// TwinCAT 3 PLC project ph_lv1_Motion
// Title: tclib_ph_lv1_motion
// Company: Poh
// Author: Poh
// ProjectVersion: 0.1.3.0
// ProgramVersion: 3.1.4020.1
// libraries:
//   Tc2_MC2, * (Beckhoff Automation GmbH)
//   tclib_ph_lv0, * (Poh)
// project tree:
//   Lv1_Motion/Class/ C_ACTUATION.TcPOU, C_ACTUATION_EXT_HOMING.TcPOU
//   Lv1_Motion/Data/ S_ACTUATION_LINK.TcDUT
//   Lv1_Motion/Interface/ IFC_ACTUATION.TcIO
// (motion and I/O tree: see PLC project ph_lv0)
// real-time tasks:
//   TASK PlcTask: cycle T#10ms, priority 20, ADS port 350
//   TASK Fast: cycle T#3ms, priority 1, ADS port 351

// ---- Lv1_Motion/Data/S_ACTUATION_LINK.TcDUT
TYPE S_ACTUATION_LINK :
STRUCT
	HARDWARE_ERROR_ID 	: UDINT;
	CALIBRATION_SENSOR	: BOOL;
	LIMIT_MINUS 		: BOOL;
	LIMIT_PLUS			: BOOL;
END_STRUCT
END_TYPE

// ---- Lv1_Motion/Interface/IFC_ACTUATION.TcIO
INTERFACE IFC_ACTUATION

PROPERTY Acceleration : LREAL
GET
END_GET
SET
END_SET
END_PROPERTY

PROPERTY Axis_Id : UDINT
GET
END_GET
END_PROPERTY

(*
	Y:2016		M:05	D:20
	D: Initiates the manual motion of the actuation device. Keep the method running for as long as manual motion is required. Terminate manual motion by calling the opposite method.
*)
METHOD Begin_Jog : RETURN_CODE
VAR_INPUT
	Towards_Positive : BOOL;
END_VAR
END_METHOD

PROPERTY Calibrate_At_Minus : BOOL
GET
END_GET
SET
END_SET
END_PROPERTY

PROPERTY Controller_Override : LREAL
GET
END_GET
SET
END_SET
END_PROPERTY

PROPERTY Current_Position : LREAL
GET
END_GET
END_PROPERTY

PROPERTY Current_Velocity : LREAL
GET
END_GET
END_PROPERTY

PROPERTY Deceleration : LREAL
GET
END_GET
SET
END_SET
END_PROPERTY

(*
	Y:2016		M:05	D:20
	D: Sets the actuation device in a de-energised state, and disable travel on both directions.
*)
METHOD Disable : RETURN_CODE
VAR_INPUT
END_VAR
END_METHOD

PROPERTY Enable : BOOL
GET
END_GET
SET
END_SET
END_PROPERTY

(*
	Y:2016		M:05	D:20
	D: Sets the actuation device in a energised state, and enable travel on both directions.
*)
METHOD Enable_All : RETURN_CODE
VAR_INPUT
END_VAR
END_METHOD

PROPERTY Enable_Bw : BOOL
GET
END_GET
SET
END_SET
END_PROPERTY

PROPERTY Enable_Fw : BOOL
GET
END_GET
SET
END_SET
END_PROPERTY

(*
	Y:2016		M:05	D:20
	D: Terminates the manual motion of the actuation device.
*)
METHOD End_Jog : RETURN_CODE
VAR_INPUT
END_VAR
END_METHOD

(*
	Y:2016		M:05	D:20
	D: Halts the actuation device.
*)
METHOD Halt : RETURN_CODE
VAR_INPUT
END_VAR
END_METHOD

(*
	Y:2016		M:05	D:20
	D: Initiates the homing sequence for the actuation device. Configure the homing behavior via the class's properties.
*)
METHOD Home : RETURN_CODE
VAR_INPUT
END_VAR
END_METHOD

PROPERTY Home_To_Limit : BOOL
GET
END_GET
SET
END_SET
END_PROPERTY

PROPERTY Is_Disabled : BOOL
GET
END_GET
END_PROPERTY

PROPERTY Is_Error : BOOL
GET
END_GET
END_PROPERTY

PROPERTY Is_Moving : BOOL
GET
END_GET
END_PROPERTY

PROPERTY Jerk : LREAL
GET
END_GET
SET
END_SET
END_PROPERTY

(*
	Y:2016		M:05	D:20
	D: Sets the actuation in motion along a direction.
*)
METHOD Move_Along : RETURN_CODE
VAR_INPUT
	Positive_Direction : BOOL;
END_VAR
END_METHOD

(*
	Y:2016		M:05	D:20
	D: Sets the actuation device in motion for a specified distance.
*)
METHOD Move_By : RETURN_CODE
VAR_INPUT
	//User defined distance to travel. Can be + or -
		Distance : LREAL;
END_VAR
END_METHOD

(*
	Y:2016		M:05	D:20
	D: Sets the actuation in motion to the target position.
*)
METHOD Move_To : RETURN_CODE
VAR_INPUT
	//User defined position to travel. Can be + or -
		POSITION : LREAL;
END_VAR
END_METHOD

(*
	Y:2016		M:05	D:20
	D: Resets the actuation device of any errors. Actuation device currently in motion will be halted.
*)
METHOD Reset : RETURN_CODE
VAR_INPUT
END_VAR
END_METHOD

PROPERTY Velocity : LREAL
GET
END_GET
SET
END_SET
END_PROPERTY

END_INTERFACE

// ---- Lv1_Motion/Class/C_ACTUATION.TcPOU
(*
	Y:2016		M:05		D:20
	T:CLASS		N:ACTUATION
	D:Class object for plc motion projects. Contains all basic necessary methods for movement. The default behavior is to home to negative limit.
*)
FUNCTION_BLOCK C_ACTUATION IMPLEMENTS IFC_ACTUATION
VAR_INPUT
END_VAR
VAR_OUTPUT
END_VAR
VAR
	//SOFTWARAE PDO LINK
		_AXIS : AXIS_REF;	
	//HARDWARE PDO LINK
		_HARDWARE_LINK	AT %I*	: S_ACTUATION_LINK;
	//MOTION MODULES
		_M_POWER 	: MC_POWER;
		_M_RESET 	: MC_RESET;
		_M_MOVEA 	: MC_MOVEABSOLUTE;
		_M_MOVER 	: MC_MOVERELATIVE;
		_M_HOME		: MC_HOME;
		_M_HALT		: MC_HALT;
		_M_MOVEEL	: MC_MoveVelocity;
		_M_JOG		: MC_JOG;
	//DYNAMICS
		_VELOCITY 		: LREAL := 10;
		_ACCELERATION 	: LREAL := 0;
		_DECELERATION 	: LREAL := 0;
		_JERK 			: LREAL := 0;
	//
		_HOME_TO_LIMIT	: BOOL := TRUE;
		_HOME_TO_MINUS	: BOOL := TRUE;
END_VAR

PROPERTY Acceleration : LREAL
GET
Acceleration := _ACCELERATION;
END_GET
SET
_ACCELERATION := ABS(Acceleration);
END_SET
END_PROPERTY

PROPERTY Axis_Id : UDINT
GET
Axis_Id := _AXIS.NcToPlc.AxisId;
END_GET
END_PROPERTY

(*
	Y:2016		M:05	D:20
	D: Initiates the manual motion of the actuation device. Keep the method running for as long as manual motion is required. Terminate manual motion by calling the opposite method.
*)
METHOD Begin_Jog : RETURN_CODE
VAR_INPUT
	Towards_Positive : BOOL;
END_VAR
_M_JOG(
	Axis:= _AXIS, 
	JogForward:= Towards_Positive, 
	JogBackwards:= NOT Towards_Positive, 
	Mode:= MC_JOGMODE_CONTINOUS, 
	Velocity:= _VELOCITY, 
	Acceleration:= _ACCELERATION, 
	Deceleration:= _DECELERATION, 
	Jerk:= _JERK);
IF _M_JOG.Error THEN
	Begin_Jog := ph_lv0.LV0_RETURNCODE.RETURN_ERROR;
ELSIF _M_JOG.CommandAborted THEN
	Begin_Jog := ph_lv0.LV0_RETURNCODE.RETURN_ERROR + 1;
ELSIF _M_JOG.Active THEN
	Begin_Jog := ph_lv0.LV0_RETURNCODE.RETURN_SUCCESS;
ELSE
	Begin_Jog := ph_lv0.LV0_RETURNCODE.RETURN_BUSY;
END_IF
END_METHOD

PROPERTY Calibrate_At_Minus : BOOL
GET
Calibrate_At_Minus := _HOME_TO_MINUS;
END_GET
SET
_HOME_TO_MINUS := Calibrate_At_Minus;
END_SET
END_PROPERTY

PROPERTY Controller_Override : LREAL
GET
VAR
	_FACTOR : LREAL := 1000000;
END_VAR
Controller_Override := (_AXIS.PlcToNc.Override / _FACTOR) * 100.0;
END_GET
SET
VAR
	_BUFFER : LREAL;
	_FACTOR : LREAL := 1000000;
END_VAR
IF Controller_Override > 100.0 THEN
	_BUFFER := 100.0;
ELSIF Controller_Override < 0.0 THEN 
	_BUFFER := 0.0;
ELSE 
	_BUFFER := Controller_Override;
END_IF
_AXIS.PlcToNc.Override := LREAL_TO_UDINT((_BUFFER/100.0) * _FACTOR);
END_SET
END_PROPERTY

PROPERTY Current_Position : LREAL
GET
Current_Position := _AXIS.NcToPlc.ActPos;
END_GET
END_PROPERTY

PROPERTY Current_Velocity : LREAL
GET
Current_Velocity := _AXIS.NcToPlc.ActVelo;
END_GET
END_PROPERTY

PROPERTY Deceleration : LREAL
GET
Deceleration := _DECELERATION;
END_GET
SET
_DECELERATION := ABS(Deceleration);
END_SET
END_PROPERTY

(*
	Y:2016		M:05	D:20
	D: Sets the actuation device in a de-energised state, and disable travel on both directions.
*)
METHOD Disable : RETURN_CODE
VAR_INPUT
END_VAR
_M_POWER(
	Axis:= _AXIS, 
	Enable:= FALSE, 
	Enable_Positive:= FALSE, 
	Enable_Negative:= FALSE, 
	Override:= 0 );

IF _M_POWER.Error THEN
	Disable := ph_lv0.LV0_RETURNCODE.RETURN_ERROR;
ELSIF NOT _M_POWER.Status THEN
	Disable := ph_lv0.LV0_RETURNCODE.RETURN_SUCCESS;
ELSE
	Disable := ph_lv0.LV0_RETURNCODE.RETURN_BUSY;
END_IF
END_METHOD

PROPERTY Enable : BOOL
GET
Enable := _AXIS.PlcToNc.ControlDWord.0;
END_GET
SET
_AXIS.PlcToNc.ControlDWord.0 := Enable;
END_SET
END_PROPERTY

(*
	Y:2016		M:05	D:20
	D: Sets the actuation device in a energised state, and enable travel on both directions.
*)
METHOD Enable_All : RETURN_CODE
VAR_INPUT
END_VAR
_M_POWER(
	Axis:= _AXIS, 
	Enable:= TRUE, 
	Enable_Positive:= TRUE, 
	Enable_Negative:= TRUE, 
	Override:= 100 );

IF _M_POWER.Error THEN
	Enable_All := ph_lv0.LV0_RETURNCODE.RETURN_ERROR;
ELSIF _M_POWER.Status THEN
	Enable_All := ph_lv0.LV0_RETURNCODE.RETURN_SUCCESS;
ELSE
	Enable_All := ph_lv0.LV0_RETURNCODE.RETURN_BUSY;
END_IF
END_METHOD

PROPERTY Enable_Bw : BOOL
GET
Enable_Bw := _AXIS.PlcToNc.ControlDWord.2;
END_GET
SET
_AXIS.PlcToNc.ControlDWord.2 := Enable_Bw;
END_SET
END_PROPERTY

PROPERTY Enable_Fw : BOOL
GET
Enable_Fw := _AXIS.PlcToNc.ControlDWord.1;
END_GET
SET
_AXIS.PlcToNc.ControlDWord.1 := Enable_Fw;
END_SET
END_PROPERTY

(*
	Y:2016		M:05	D:20
	D: Terminates the manual motion of the actuation device.
*)
METHOD End_Jog : RETURN_CODE
VAR_INPUT
END_VAR
_M_JOG(
	Axis:= _AXIS, 
	JogForward:= FALSE, 
	JogBackwards:= FALSE);
IF _M_JOG.Error THEN
	End_Jog := ph_lv0.LV0_RETURNCODE.RETURN_ERROR;
ELSIF _M_JOG.CommandAborted THEN
	End_Jog := ph_lv0.LV0_RETURNCODE.RETURN_ERROR + 1;
ELSIF _M_JOG.Done THEN
	End_Jog := ph_lv0.LV0_RETURNCODE.RETURN_SUCCESS;
ELSE
	End_Jog := ph_lv0.LV0_RETURNCODE.RETURN_BUSY;
END_IF
END_METHOD

(*
	Y:2016		M:05	D:20
	D: Halts the actuation device.
*)
METHOD Halt : RETURN_CODE
VAR_INPUT
END_VAR
_M_HALT(
	Axis:= _AXIS, 
	Execute:= TRUE, 
	Deceleration:= _DECELERATION, 
	Jerk:= _JERK);
IF _M_HALT.Error THEN
	_M_HALT(
		Axis:=_AXIS,
		Execute:=FALSE);
	Halt:=ph_lv0.LV0_RETURNCODE.RETURN_ERROR;
ELSIF _M_HALT.CommandAborted THEN
	_M_HALT(
		Axis:=_AXIS,
		Execute:=FALSE);
	Halt:=ph_lv0.LV0_RETURNCODE.RETURN_ERROR + 1;
ELSIF _M_HALT.Done THEN
	_M_HALT(
		Axis:=_AXIS,
		Execute:=FALSE);
	Halt:=ph_lv0.LV0_RETURNCODE.RETURN_SUCCESS;
ELSE
	Halt:=ph_lv0.LV0_RETURNCODE.RETURN_BUSY;
END_IF
END_METHOD

(*
	Y:2016		M:05	D:20
	D: Initiates the homing sequence for the actuation device. Configure the homing behavior via the class's properties.
*)
METHOD Home : RETURN_CODE
VAR_INPUT
END_VAR
VAR
	_CALIBRATION_FLAG : BOOL;
END_VAR
IF _HOME_TO_LIMIT THEN
	IF _HOME_TO_MINUS THEN
		_CALIBRATION_FLAG := THIS^._HARDWARE_LINK.LIMIT_MINUS;
	ELSE
		_CALIBRATION_FLAG := THIS^._HARDWARE_LINK.LIMIT_PLUS;
	END_IF
ELSE
	_CALIBRATION_FLAG := THIS^._HARDWARE_LINK.CALIBRATION_SENSOR;
END_IF
_M_HOME(
	Axis:= _AXIS, 
	Execute:= TRUE, 
	bCalibrationCam:= _CALIBRATION_FLAG);
IF _M_HOME.Error THEN
	_M_HOME(
		Axis:= _AXIS, 
		Execute:= FALSE);
	Home := ph_lv0.LV0_RETURNCODE.RETURN_ERROR;
ELSIF _M_HOME.CommandAborted THEN
	_M_HOME(
		Axis:= _AXIS, 
		Execute:= FALSE);
	Home := ph_lv0.LV0_RETURNCODE.RETURN_ERROR + 1;
ELSIF _M_HOME.Done THEN
	_M_HOME(
		Axis:= _AXIS, 
		Execute:= FALSE);
	Home := ph_lv0.LV0_RETURNCODE.RETURN_SUCCESS;
ELSE
	Home := ph_lv0.LV0_RETURNCODE.RETURN_BUSY;
END_IF
END_METHOD

PROPERTY Home_To_Limit : BOOL
GET
Home_To_Limit := _HOME_TO_LIMIT;
END_GET
SET
_HOME_TO_LIMIT := Home_To_Limit;
END_SET
END_PROPERTY

PROPERTY Is_Disabled : BOOL
GET
_AXIS.ReadStatus();
Is_Disabled := _AXIS.Status.Disabled;
END_GET
END_PROPERTY

PROPERTY Is_Error : BOOL
GET
_AXIS.ReadStatus();
Is_Error := _AXIS.Status.Error;
END_GET
END_PROPERTY

PROPERTY Is_Moving : BOOL
GET
_AXIS.ReadStatus();
Is_Moving := _AXIS.Status.Moving;
END_GET
END_PROPERTY

PROPERTY Jerk : LREAL
GET
Jerk := _JERK;
END_GET
SET
_JERK := ABS(Jerk);
END_SET
END_PROPERTY

(*
	Y:2016		M:05	D:20
	D: Sets the actuation in motion along a direction.
*)
METHOD Move_Along : RETURN_CODE
VAR_INPUT
	Positive_Direction : BOOL;
END_VAR
VAR
	_DIRECTION : MC_Direction;
END_VAR
IF Positive_Direction THEN
	_DIRECTION := MC_Direction.MC_Positive_Direction;
ELSE
	_DIRECTION := MC_Direction.MC_Negative_Direction;
END_IF
_M_MOVEEL(
	Axis:= _AXIS, 
	Execute:= TRUE, 
	Velocity:= _VELOCITY, 
	Acceleration:= _ACCELERATION, 
	Deceleration:= _DECELERATION, 
	Jerk:= _JERK, 
	Direction:= _DIRECTION);
IF _M_MOVEEL.Error THEN
	_M_MOVEEL(
		Axis:= _AXIS, 
		Execute:= FALSE); 
	Move_Along := ph_lv0.LV0_RETURNCODE.RETURN_ERROR;
ELSIF _M_MOVEEL.CommandAborted THEN
	_M_MOVEEL(
		Axis:= _AXIS, 
		Execute:= FALSE);
	Move_Along := ph_lv0.LV0_RETURNCODE.RETURN_ERROR + 1;
ELSIF _M_MOVEEL.InVelocity THEN
	_M_MOVEEL(
		Axis:= _AXIS, 
		Execute:= FALSE);
	Move_Along := ph_lv0.LV0_RETURNCODE.RETURN_SUCCESS;
ELSE
	Move_Along := ph_lv0.LV0_RETURNCODE.RETURN_BUSY;
END_IF
END_METHOD

(*
	Y:2016		M:05	D:20
	D: Sets the actuation device in motion for a specified distance.
*)
METHOD Move_By : RETURN_CODE
VAR_INPUT
	//User defined distance to travel. Can be + or -
		Distance : LREAL;
END_VAR
_M_MOVER(
	Axis:= _AXIS, 
	Execute:= TRUE, 
	Distance:= Distance, 
	Velocity:= _VELOCITY, 
	Acceleration:= _ACCELERATION, 
	Deceleration:= _DECELERATION, 
	Jerk:= _JERK);
	
IF _M_MOVER.Error THEN
	_M_MOVER(
		Axis:= _AXIS, 
		Execute:= FALSE);
	Move_By := ph_lv0.LV0_RETURNCODE.RETURN_ERROR;
ELSIF _M_MOVER.CommandAborted THEN
	_M_MOVER(
		Axis:= _AXIS, 
		Execute:= FALSE);
	Move_By := ph_lv0.LV0_RETURNCODE.RETURN_ERROR + 1;
ELSIF _M_MOVER.Done THEN
	_M_MOVER(
		Axis:= _AXIS, 
		Execute:= FALSE);
	Move_By := ph_lv0.LV0_RETURNCODE.RETURN_SUCCESS;
ELSE
	Move_By := ph_lv0.LV0_RETURNCODE.RETURN_BUSY;	
END_IF
END_METHOD

(*
	Y:2016		M:05	D:20
	D: Sets the actuation in motion to the target position.
*)
METHOD Move_To : RETURN_CODE
VAR_INPUT
	//User defined position to travel. Can be + or -
		POSITION : LREAL;
END_VAR
_M_MOVEA(
	Axis:= _AXIS, 
	Execute:= TRUE, 
	Position:= POSITION, 
	Velocity:= _VELOCITY, 
	Acceleration:= _ACCELERATION, 
	Deceleration:= _DECELERATION, 
	Jerk:= _JERK);
IF _M_MOVEA.Error THEN
	_M_MOVEA(
		Axis:= _AXIS, 
		Execute:= FALSE);
	Move_To := ph_lv0.LV0_RETURNCODE.RETURN_ERROR;
ELSIF _M_MOVEA.CommandAborted THEN
	_M_MOVEA(
		Axis:= _AXIS, 
		Execute:= FALSE);
	Move_To := ph_lv0.LV0_RETURNCODE.RETURN_ERROR + 1;
ELSIF _M_MOVEA.Done THEN
	_M_MOVEA(
		Axis:= _AXIS, 
		Execute:= FALSE);
	Move_To := ph_lv0.LV0_RETURNCODE.RETURN_SUCCESS;
ELSE
	Move_To := ph_lv0.LV0_RETURNCODE.RETURN_BUSY;	
END_IF
END_METHOD

(*
	Y:2016		M:05	D:20
	D: Resets the actuation device of any errors. Actuation device currently in motion will be halted.
*)
METHOD Reset : RETURN_CODE
VAR_INPUT
END_VAR
//RESET OTHER FUNCTION BLOCKS
	_M_MOVEA(
		Axis:= _AXIS,
		Execute:= FALSE);
	_M_MOVER(
		Axis:= _AXIS, 
		Execute:= FALSE);
	_M_MOVEEL(
		Axis:= _AXIS, 
		Execute:= FALSE);
	_M_HALT(
		Axis:= _AXIS, 
		Execute:= FALSE);
	_M_HOME(
		Axis:= _AXIS, 
		Execute:= FALSE);
//EXECUTE RESET
	_M_RESET(
		Axis:= _AXIS, 
		Execute:= TRUE);
	IF _M_RESET.Error THEN
		_M_RESET(
			Axis:= _AXIS, 
			Execute:= FALSE);
		Reset := ph_lv0.LV0_RETURNCODE.RETURN_ERROR;
	ELSIF _M_RESET.Done AND NOT _M_RESET.Busy THEN
		_M_RESET(
			Axis:= _AXIS, 
			Execute:= FALSE);
		Reset := ph_lv0.LV0_RETURNCODE.RETURN_SUCCESS;
	ELSE
		Reset := ph_lv0.LV0_RETURNCODE.RETURN_BUSY;	
	END_IF
END_METHOD

PROPERTY Velocity : LREAL
GET
Velocity := _VELOCITY;
END_GET
SET
_VELOCITY := ABS(Velocity);
END_SET
END_PROPERTY

END_FUNCTION_BLOCK

// ---- Lv1_Motion/Class/C_ACTUATION_EXT_HOMING.TcPOU
FUNCTION_BLOCK C_ACTUATION_EXT_HOMING EXTENDS C_ACTUATION
VAR_INPUT
END_VAR
VAR_OUTPUT
END_VAR
VAR
	_HardStopCalibration	: BOOL := FALSE;
	_HardStopTol			: LREAL := 5.0;
END_VAR

PROPERTY Calibrate_At_Hardstop : BOOL
GET
Calibrate_At_Hardstop := _HardStopCalibration;
END_GET
SET
_HardStopCalibration := Calibrate_At_Hardstop;
END_SET
END_PROPERTY

PROPERTY Hardstop_Tolerance : LREAL
GET
Hardstop_Tolerance := _HardStopTol;
END_GET
SET
 _HardStopTol := Hardstop_Tolerance;
END_SET
END_PROPERTY

{attribute '''NORMAL__COMMENT' := '
	Y:2016		M:05	D:20
	D: Initiates the homing sequence for the actuation device. Configure the homing behavior via the class's properties.
'}
(*
	Y:2016		M:05	D:20
	D: Initiates the homing sequence for the actuation device. Configure the homing behavior via the class's properties.
*)
(*
	Y:2016		M:06	D:03
	D: Initiates the homing sequence for the actuation device. Configure the homing behavior via the class's properties.
	EXT: Uses the Use_Hard_Stop option to calibrate the homing sequence
*)
METHOD Home : ph_lv0.RETURN_CODE
VAR
	_CALIBRATION_FLAG : BOOL;
END_VAR
IF _HardStopCalibration THEN
	_CALIBRATION_FLAG := ABS(_AXIS.NcToPlc.PosDiff) > _HardStopTol;
ELSE 
	IF _HOME_TO_LIMIT THEN
		IF _HOME_TO_MINUS THEN
			_CALIBRATION_FLAG := THIS^._HARDWARE_LINK.LIMIT_MINUS;
		ELSE
			_CALIBRATION_FLAG := THIS^._HARDWARE_LINK.LIMIT_PLUS;
		END_IF
	ELSE
		_CALIBRATION_FLAG := THIS^._HARDWARE_LINK.CALIBRATION_SENSOR;
	END_IF
END_IF
_M_HOME(
	Axis:= _AXIS, 
	Execute:= TRUE, 
	bCalibrationCam:= _CALIBRATION_FLAG);
IF _M_HOME.Error THEN
	_M_HOME(
		Axis:= _AXIS, 
		Execute:= FALSE);
	Home := ph_lv0.LV0_RETURNCODE.RETURN_ERROR;
ELSIF _M_HOME.CommandAborted THEN
	_M_HOME(
		Axis:= _AXIS, 
		Execute:= FALSE);
	Home := ph_lv0.LV0_RETURNCODE.RETURN_ERROR + 1;
ELSIF _M_HOME.Done THEN
	_M_HOME(
		Axis:= _AXIS, 
		Execute:= FALSE);
	Home := ph_lv0.LV0_RETURNCODE.RETURN_SUCCESS;
ELSE
	Home := ph_lv0.LV0_RETURNCODE.RETURN_BUSY;
END_IF
END_METHOD

END_FUNCTION_BLOCK
